RoboDK station: main for aircraftCOPY.rdk

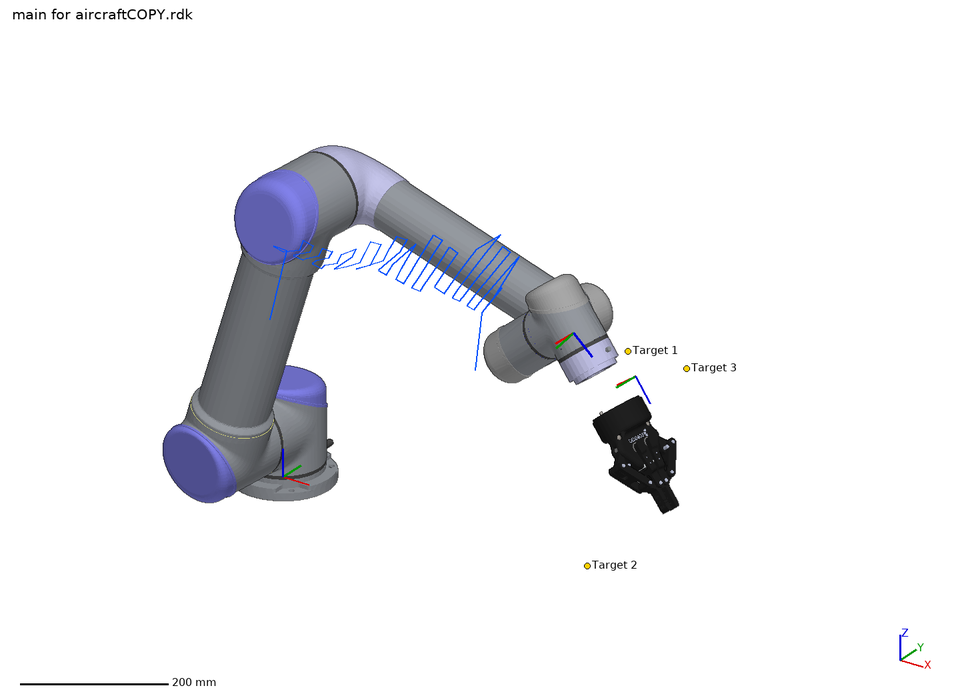
[picture v0: the station drawn from its stored meshes, robots at their saved joint values, targets as dots, program paths as lines]
Station main. Poses are relative to the parent item; angles as X-Y-Z fixed-axis rotations.
  - frame UR5 Base at (0, 0, 0) mm
    - robot UR5: 6 axes, payload 5 kg, reach 850 mm, repeatability 0.1 mm, weight 18.4 kg
        modified DH rows (alpha deg, a mm, theta deg, d mm): 0, 0, 0, 89.2; 90, 0, 180, 0; 0, 425, 0, 0; 0, 392.43, 0, 109; -90, 0, 0, 93.65; 90, 0, 180, 82
        joint limits [-360, -360, -360, -360, -360, -360] to [360, 360, 360, 360, 360, 360]; home [0, -90, -90, 0, 90, 0]; saved at [-4.126, -107.813, -86.6, -35.896, 88.406, -3.183]
      - tool Gripper RobotiQ 85 Fully closed, TCP at (0, 0, 266.2) mm, size 121.5 x 75 x 160.2 mm
      - frame Object at (8, -67.5, 31) mm
    - target Target 1 (Cartesian target) at (643.45, -109, 411.64) mm, rotated rx -90 ry 0 rz -90 deg; joints [0, -86.624, -123.251, 29.876, 90, 0] of UR5
    - target Target 2 (Cartesian target) at (575.78, -109, 70.86) mm, rotated rx -135 ry 0 rz -90 deg; joints [0, -90, -135, 0, 90, 0] of UR5
    - target Target 3 (Cartesian target) at (739.63, -109, 412.97) mm, rotated rx -105 ry 0 rz -90 deg; joints [0, -90, -105, 0, 90, 0] of UR5
    - frame Object at (559.36, -117, 419.3) mm, rotated rx -132.29 ry 0 rz -90 deg
      - object cloud_8 at (0, 0, 0) mm
  - program Path1 (108 instructions, listed below)
  - machining project Path1 settings: rotZ(0) | rotX(0)*rotY(0) | rotZ(0) | onStart | onPathStart | onApproach | onPoint | onRetract | onFinish | SetRPM(%1) | SetTool(%1) | Extruder(%1) | default | default | OutOnMov(%1) | OutOffMov(%1) | onPathFinish | M_RunCode(%1)
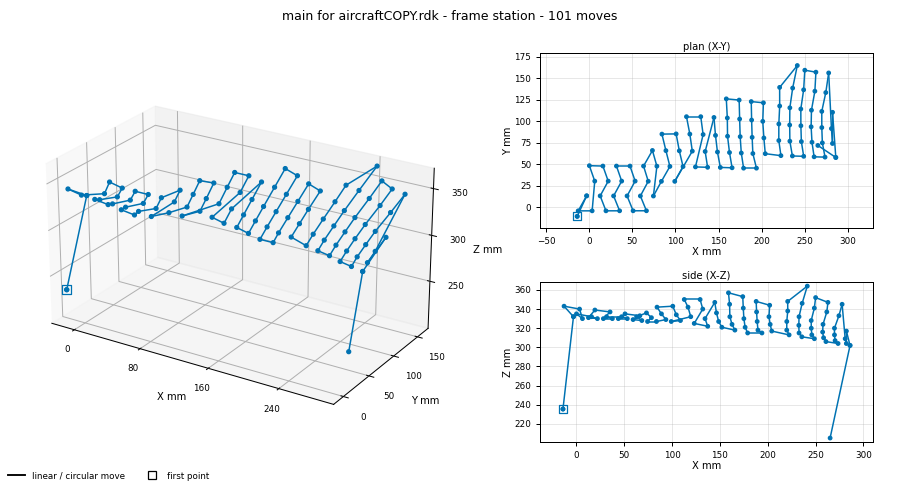
[picture p0: tool path of main for aircraftCOPY.rdk in frame station, 101 of 101 moves have a stored position in this frame; points joined in program order, loops and branches not executed]

--- program Path1 (robot UR5) ---
  Smooth(5)
  Set Ref.: UR5 Base
  Set Tool: Gripper RobotiQ 85 Fully closed
  Show Gripper RobotiQ 85 Fully closed
  Set speed (5.0 mm/s)
  MoveJ 1 to (-14.04, -10.4, 235.49) mm, rotated rx -13.93 ry 6.12 rz -1.51 deg; joints [4.658, -99.481, -81.097, -56.074, 81.119, 3.913]
  MoveL 2 to (-14.04, -10.4, 235.49) mm, rotated rx -13.93 ry 6.12 rz -1.51 deg; joints [4.658, -99.481, -81.097, -56.074, 81.119, 3.913]
  MoveL 3 to (-3.06, 13.38, 332) mm, rotated rx -13.93 ry 6.12 rz -1.51 deg; joints [3.175, -108.37, -82.037, -46.06, 81.936, 2.662]
  MoveL 4 to (-3.06, 13.38, 332) mm, rotated rx -13.93 ry 6.12 rz -1.51 deg; joints [3.175, -108.37, -82.037, -46.06, 81.936, 2.662]
  Set speed (5.0 mm/s)
  MoveL 5 to (-12.91, -4.04, 343) mm, rotated rx -32.27 ry 3.58 rz -2.26 deg; joints [2.431, -124.577, -46.301, -83.798, 85.122, 2.351]
  MoveL 6 to (3.3, -4, 340) mm, rotated rx -29.46 ry 5.28 rz -2.98 deg; joints [2.075, -121.423, -52.584, -77.822, 83.29, 1.983]
  MoveL 7 to (6.33, 30.48, 330) mm, rotated rx 2.3 ry 4.12 rz 0.17 deg; joints [1.192, -104.072, -102.448, -13.533, 84.96, 0.769]
  MoveL 8 to (0.08, 48.39, 335) mm, rotated rx 9.26 ry 5.03 rz 0.82 deg; joints [2.717, -105.068, -110.917, 2.753, 82.63, 1.494]
  MoveL 9 to (15.8, 47.96, 332) mm, rotated rx 8.64 ry 2.64 rz 0.4 deg; joints [-0.895, -105.14, -109.708, 1.212, 88.073, -0.496]
  MoveL 10 to (21.95, 30.48, 330) mm, rotated rx 1.48 ry 1.8 rz 0.05 deg; joints [-2.088, -104.786, -100.703, -15.298, 89.78, -1.364]
  MoveL 11 to (12.62, 13.34, 331) mm, rotated rx -12.78 ry 2.95 rz -0.67 deg; joints [-0.216, -108.437, -82.477, -44.133, 87.1, -0.177]
  MoveL 12 to (19.34, -3.99, 339) mm, rotated rx -27.21 ry 3.75 rz -1.93 deg; joints [-0.143, -119.939, -55.839, -73.653, 85.831, -0.134]
  MoveL 13 to (35.18, -3.97, 337) mm, rotated rx -25.88 ry 3.5 rz -1.7 deg; joints [-1.638, -119.083, -57.679, -71.257, 86.718, -1.522]
  MoveL 14 to (28.2, 13.3, 330) mm, rotated rx -11.29 ry 2.61 rz -0.52 deg; joints [-1.946, -108.209, -83.758, -41.541, 88.497, -1.566]
  MoveL 15 to (37.57, 30.48, 330) mm, rotated rx 1.89 ry 1.74 rz 0.06 deg; joints [-3.839, -105.297, -100.404, -14.689, 91.184, -2.488]
  MoveL 16 to (31.52, 47.96, 332) mm, rotated rx 6.96 ry 1.23 rz 0.15 deg; joints [-3.717, -105.465, -107.483, -2.398, 91.793, -2.15]
  MoveL 17 to (47.23, 47.96, 332) mm, rotated rx 8.92 ry 1.1 rz 0.17 deg; joints [-5.68, -106.487, -108.129, 1.171, 93.63, -3.127]
  MoveL 18 to (53.2, 30.48, 330) mm, rotated rx 3.33 ry 3.03 rz 0.18 deg; joints [-4.727, -105.67, -101.292, -11.942, 90.643, -2.971]
  MoveL 19 to (43.82, 13.3, 330) mm, rotated rx -9.75 ry 3.74 rz -0.64 deg; joints [-2.827, -107.971, -85.284, -38.649, 87.952, -2.229]
  MoveL 20 to (50.83, -3.94, 335) mm, rotated rx -26.54 ry 2.66 rz -1.33 deg; joints [-3.395, -120.113, -55.49, -73.063, 88.259, -3.166]
  MoveL 21 to (66.29, -3.92, 333) mm, rotated rx -26.5 ry 0.34 rz -0.17 deg; joints [-5.97, -121.072, -53.703, -74.084, 91.773, -5.567]
  MoveL 22 to (59.27, 13.26, 329) mm, rotated rx -8.2 ry 4.18 rz -0.6 deg; joints [-4.126, -107.813, -86.6, -35.896, 88.406, -3.183]
  MoveL 23 to (68.4, 30.3, 328) mm, rotated rx 4.71 ry 3.77 rz 0.31 deg; joints [-5.958, -105.952, -102.01, -9.54, 90.942, -3.631]
  MoveL 24 to (62.95, 47.96, 332) mm, rotated rx 11.37 ry 2.76 rz 0.56 deg; joints [-6.391, -107.482, -109.437, 5.996, 92.664, -3.283]
  MoveL 25 to (73.25, 66.03, 336) mm, rotated rx 17.27 ry 1.87 rz 0.58 deg; joints [-8.642, -111.204, -114.03, 20.082, 95.874, -3.664]
  MoveL 26 to (78.43, 47.81, 331) mm, rotated rx 12.53 ry 3.11 rz 0.69 deg; joints [-7.991, -108.278, -109.451, 7.928, 93.753, -3.968]
  MoveL 27 to (74.39, 13.18, 327) mm, rotated rx -4.76 ry 3.26 rz -0.27 deg; joints [-6.351, -107.433, -89.554, -29.969, 91.059, -4.644]
  MoveL 28 to (83.67, 30.21, 327) mm, rotated rx 6.61 ry 3.96 rz 0.46 deg; joints [-7.59, -106.614, -102.837, -6.179, 92.179, -4.424]
  MoveL 29 to (93.53, 47.52, 329) mm, rotated rx 13.66 ry 4.79 rz 1.16 deg; joints [-8.579, -108.731, -109.835, 9.966, 92.601, -4.11]
  MoveL 30 to (88.89, 65.84, 335) mm, rotated rx 18.59 ry 2.63 rz 0.88 deg; joints [-10.002, -112.249, -113.92, 22.315, 96.386, -4.032]
  MoveL 31 to (84.27, 85.02, 342) mm, rotated rx 19.46 ry 0.64 rz 0.23 deg; joints [-11.204, -114.4, -115.675, 26.899, 99.636, -4.386]
  MoveL 32 to (100.76, 85.27, 343) mm, rotated rx 22.25 ry 2.56 rz 1.05 deg; joints [-11.8, -116.671, -116.019, 32.433, 98.32, -4.065]
  MoveL 33 to (104.44, 65.64, 334) mm, rotated rx 20.16 ry 4.48 rz 1.64 deg; joints [-10.489, -113.289, -114.187, 25.277, 94.948, -3.958]
  MoveL 34 to (108.77, 47.38, 328) mm, rotated rx 15.72 ry 6.99 rz 1.96 deg; joints [-8.804, -109.718, -110.698, 13.955, 90.618, -3.942]
  MoveL 35 to (99.15, 30.21, 327) mm, rotated rx 8.68 ry 5.48 rz 0.83 deg; joints [-8.36, -107.362, -103.956, -2.166, 91.429, -4.622]
  MoveL 36 to (119.53, 65.25, 332) mm, rotated rx 21.76 ry 7.28 rz 2.9 deg; joints [-10.132, -114.088, -114.701, 28.264, 91.652, -3.57]
  MoveL 37 to (116.65, 85.02, 342) mm, rotated rx 23.97 ry 4.72 rz 2.09 deg; joints [-12.039, -117.925, -116.146, 35.627, 96.264, -3.799]
  MoveL 38 to (112.76, 105.23, 350) mm, rotated rx 22.75 ry 2.4 rz 1.01 deg; joints [-13.632, -119.241, -116.861, 36.235, 100.237, -4.599]
  MoveL 39 to (129.32, 105.23, 350) mm, rotated rx 25.49 ry 5.83 rz 2.77 deg; joints [-12.898, -121.304, -117.349, 41.728, 95.891, -3.75]
  MoveL 40 to (132.07, 84.52, 340) mm, rotated rx 25.16 ry 7.46 rz 3.49 deg; joints [-11.683, -118.575, -116.325, 37.699, 92.926, -3.469]
  MoveL 41 to (123.16, 46.95, 325) mm, rotated rx 17.31 ry 8.78 rz 2.72 deg; joints [-9.209, -110.364, -111.216, 16.734, 89.155, -3.906]
  MoveL 42 to (137.27, 46.51, 322) mm, rotated rx 18.11 ry 9.74 rz 3.17 deg; joints [-10.188, -110.797, -111.09, 17.851, 89.059, -4.198]
  MoveL 43 to (134.43, 64.85, 330) mm, rotated rx 21.94 ry 8.91 rz 3.57 deg; joints [-10.654, -114.25, -114.327, 28.246, 90.392, -3.735]
  MoveL 44 to (144.64, 104.33, 347) mm, rotated rx 27.45 ry 6.48 rz 3.35 deg; joints [-14.285, -122.842, -116.779, 44.62, 96.51, -3.692]
  MoveL 45 to (146.42, 83.53, 336) mm, rotated rx 26.11 ry 8.64 rz 4.21 deg; joints [-12.502, -119.014, -116.077, 38.811, 92.396, -3.528]
  MoveL 46 to (148.69, 64.26, 327) mm, rotated rx 21.87 ry 9.27 rz 3.7 deg; joints [-12.115, -114.309, -113.603, 27.514, 91.369, -4.26]
  MoveL 47 to (152.04, 46.37, 321) mm, rotated rx 18.81 ry 9.71 rz 3.29 deg; joints [-11.955, -111.655, -110.45, 18.745, 90.723, -4.788]
  MoveL 48 to (165.67, 45.93, 318) mm, rotated rx 18.23 ry 9.46 rz 3.1 deg; joints [-13.74, -111.641, -109.321, 17.009, 92.603, -5.619]
  MoveL 49 to (162.66, 63.67, 324) mm, rotated rx 22.01 ry 9.27 rz 3.72 deg; joints [-13.823, -114.576, -112.803, 27.09, 92.981, -4.826]
  MoveL 50 to (160.39, 82.53, 332) mm, rotated rx 26.15 ry 8.57 rz 4.18 deg; joints [-14.321, -119.011, -115.28, 38.024, 94.217, -4.029]
  MoveL 51 to (160.14, 103.73, 345) mm, rotated rx 29.01 ry 7.31 rz 4.04 deg; joints [-15.477, -124.202, -116.052, 46.772, 96.704, -3.605]
  MoveL 52 to (158.95, 125.93, 357) mm, rotated rx 25.77 ry 6.33 rz 3.05 deg; joints [-16.373, -124.524, -116.673, 44.444, 98.668, -4.696]
  MoveL 53 to (173.88, 124.52, 353) mm, rotated rx 25.79 ry 10.53 rz 5.05 deg; joints [-14.709, -123.729, -117.264, 44.369, 92.422, -4.254]
  MoveL 54 to (174.43, 102.53, 341) mm, rotated rx 29.39 ry 9.23 rz 5.16 deg; joints [-15.613, -124.047, -115.912, 46.829, 94.645, -3.565]
  MoveL 55 to (175.05, 82.04, 330) mm, rotated rx 26.13 ry 8.93 rz 4.35 deg; joints [-15.808, -119.248, -114.366, 37.298, 95.246, -4.456]
  MoveL 56 to (176.35, 63.08, 321) mm, rotated rx 21.27 ry 8.37 rz 3.24 deg; joints [-16.144, -114.531, -111.386, 24.811, 96.094, -5.818]
  MoveL 57 to (179.02, 45.5, 315) mm, rotated rx 17.33 ry 7.76 rz 2.41 deg; joints [-16.496, -111.814, -107.484, 14.249, 96.84, -6.975]
  MoveL 58 to (193.93, 45.5, 315) mm, rotated rx 15.83 ry 5.39 rz 1.53 deg; joints [-19.64, -112.544, -104.549, 10.067, 101.967, -8.828]
  MoveL 59 to (189.76, 62.49, 318) mm, rotated rx 20.07 ry 7.01 rz 2.55 deg; joints [-18.678, -114.416, -109.502, 21.397, 99.823, -7.106]
  MoveL 60 to (188.94, 81.29, 327) mm, rotated rx 24.51 ry 8.87 rz 4.02 deg; joints [-17.525, -118.312, -113.096, 33.447, 96.94, -5.406]
  MoveL 61 to (188.34, 101.33, 337) mm, rotated rx 28.37 ry 10.38 rz 5.56 deg; joints [-16.395, -122.948, -115.43, 44.227, 94.131, -4.042]
  MoveL 62 to (187.89, 122.75, 348) mm, rotated rx 25.98 ry 12.27 rz 5.91 deg; joints [-15.025, -123.348, -117.013, 43.906, 90.8, -4.333]
  MoveL 63 to (202.02, 121.34, 344) mm, rotated rx 26.28 ry 11.02 rz 5.39 deg; joints [-17.837, -123.694, -115.725, 43.214, 94.876, -5.018]
  MoveL 64 to (201.26, 99.82, 332) mm, rotated rx 27.33 ry 10.65 rz 5.46 deg; joints [-17.822, -121.884, -114.696, 41.39, 95.245, -4.702]
  MoveL 65 to (202.54, 80.55, 324) mm, rotated rx 22.52 ry 9.94 rz 4.09 deg; joints [-18.273, -117.028, -112.036, 29.179, 96.45, -6.232]
  MoveL 66 to (204.17, 62.3, 317) mm, rotated rx 18.16 ry 8.15 rz 2.66 deg; joints [-19.337, -113.803, -108.009, 17.452, 99.078, -7.939]
  MoveL 67 to (222.34, 60.03, 313) mm, rotated rx 14.21 ry 10.15 rz 2.56 deg; joints [-19.65, -112.166, -105.317, 9.466, 96.895, -9.244]
  MoveL 68 to (219.87, 77.55, 318) mm, rotated rx 18.99 ry 11.07 rz 3.78 deg; joints [-19.319, -114.796, -109.944, 21.46, 96.054, -7.674]
  MoveL 69 to (219.9, 96.77, 327) mm, rotated rx 25.69 ry 11.78 rz 5.61 deg; joints [-19.141, -120.51, -113.4, 37.111, 95.29, -5.582]
  MoveL 70 to (220.9, 117.63, 338) mm, rotated rx 27.73 ry 10.98 rz 5.72 deg; joints [-20.124, -124.595, -114.319, 44.049, 97.089, -5.184]
  MoveL 71 to (220.84, 139.23, 348) mm, rotated rx 31.61 ry 8.27 rz 5.06 deg; joints [-22.652, -130.842, -113.821, 53.503, 102.558, -4.337]
  MoveL 72 to (241.33, 164.59, 364) mm, rotated rx 35.26 ry 21.55 rz 14.56 deg; joints [-13.058, -135.826, -115.512, 62.282, 77.077, -2.264]
  MoveL 73 to (235.95, 138.43, 346) mm, rotated rx 31.94 ry 10.5 rz 6.48 deg; joints [-22.483, -130.861, -113.54, 53.548, 99.763, -4.227]
  MoveL 74 to (232.69, 115.54, 332) mm, rotated rx 28.97 ry 12.2 rz 6.68 deg; joints [-20.555, -124.887, -114.124, 45.319, 96.085, -4.911]
  MoveL 75 to (232.5, 95.59, 323) mm, rotated rx 24.2 ry 12.01 rz 5.34 deg; joints [-20.468, -119.484, -112.318, 33.541, 96.302, -6.46]
  MoveL 76 to (232.71, 76.82, 315) mm, rotated rx 17.53 ry 11.11 rz 3.48 deg; joints [-20.671, -114.346, -108.378, 17.969, 97.14, -8.681]
  MoveL 77 to (235.64, 59.65, 311) mm, rotated rx 12.24 ry 10.4 rz 2.24 deg; joints [-20.74, -111.961, -103.23, 5.235, 97.351, -10.365]
  MoveL 78 to (248.75, 59.26, 309) mm, rotated rx 12.05 ry 9.71 rz 2.06 deg; joints [-22.542, -112.61, -101.691, 3.921, 99.584, -11.351]
  MoveL 79 to (246.05, 76.33, 313) mm, rotated rx 16.26 ry 10.32 rz 2.99 deg; joints [-22.593, -114.428, -106.368, 14.602, 99.578, -9.94]
  MoveL 80 to (245.49, 94.7, 320) mm, rotated rx 22.41 ry 11.51 rz 4.7 deg; joints [-22.316, -118.687, -110.672, 29.268, 98.548, -7.676]
  MoveL 81 to (245.42, 114.15, 328) mm, rotated rx 28.59 ry 12.25 rz 6.59 deg; joints [-22.065, -124.555, -113.171, 43.627, 97.517, -5.409]
  MoveL 82 to (248.69, 136.43, 341) mm, rotated rx 30.93 ry 11.5 rz 6.81 deg; joints [-23.225, -129.548, -113.211, 50.878, 99.389, -4.786]
  MoveL 83 to (250.04, 159.16, 352) mm, rotated rx 26.25 ry 18.79 rz 9.03 deg; joints [-17.787, -127.605, -116.462, 47.664, 86.247, -5.294]
  MoveL 84 to (262.92, 156.9, 347) mm, rotated rx 21.2 ry 15.74 rz 6.01 deg; joints [-21.942, -124.051, -114.454, 37.527, 93.638, -8.034]
  MoveL 85 to (261.72, 134.83, 337) mm, rotated rx 31 ry 11.54 rz 6.85 deg; joints [-24.728, -129.529, -112.168, 49.83, 100.814, -5.073]
  MoveL 86 to (257.76, 112.76, 324) mm, rotated rx 27.1 ry 12.19 rz 6.17 deg; joints [-23.593, -123.475, -112.082, 39.969, 99.09, -6.354]
  MoveL 87 to (257.38, 93.52, 316) mm, rotated rx 20.85 ry 12.11 rz 4.57 deg; joints [-23.182, -117.732, -109.535, 25.67, 98.637, -8.55]
  MoveL 88 to (258.36, 75.6, 310) mm, rotated rx 14.7 ry 11.57 rz 3.01 deg; joints [-22.947, -113.864, -105.096, 11.402, 98.422, -10.624]
  MoveL 89 to (260.82, 58.69, 306) mm, rotated rx 11.48 ry 10.6 rz 2.14 deg; joints [-23.175, -112.649, -100.685, 2.498, 99.145, -11.851]
  MoveL 90 to (273.51, 58.3, 304) mm, rotated rx 10.15 ry 11.57 rz 2.06 deg; joints [-23.693, -112.669, -99.127, -0.18, 98.385, -12.554]
  MoveL 91 to (270.4, 74.87, 307) mm, rotated rx 13.4 ry 11.33 rz 2.68 deg; joints [-24.269, -113.79, -103.28, 8.123, 99.653, -11.719]
  MoveL 92 to (269.75, 92.63, 313) mm, rotated rx 19.54 ry 12.42 rz 4.37 deg; joints [-24.263, -117.246, -108.159, 22.511, 99.222, -9.449]
  MoveL 93 to (269.73, 111.36, 320) mm, rotated rx 25.95 ry 12.08 rz 5.82 deg; joints [-25.067, -122.725, -110.92, 36.872, 100.629, -7.22]
  MoveL 94 to (274.38, 133.23, 333) mm, rotated rx 32.33 ry 11.69 rz 7.31 deg; joints [-26.013, -130.482, -111.059, 50.918, 101.818, -4.774]
  MoveL 95 to (277.73, 156, 345) mm, rotated rx 16.02 ry 10.84 rz 3.09 deg; joints [-26.843, -121.881, -110.129, 25.286, 102.813, -11.95]
  MoveL 96 to (280.94, 91.44, 309) mm, rotated rx 17.97 ry 12.11 rz 3.89 deg; joints [-25.625, -116.644, -106.509, 18.613, 100.652, -10.61]
  MoveL 97 to (282.15, 74.13, 304) mm, rotated rx 12.59 ry 11.89 rz 2.63 deg; joints [-25.048, -113.779, -102.009, 6.089, 99.639, -12.391]
  MoveL 98 to (282.21, 110.32, 317) mm, rotated rx 25.69 ry 12.39 rz 5.89 deg; joints [-26.213, -122.71, -109.865, 35.49, 101.381, -7.676]
  MoveL 99 to (286.01, 57.92, 302) mm, rotated rx 8.38 ry 11.9 rz 1.74 deg; joints [-24.523, -112.802, -96.959, -3.897, 98.433, -13.603]
  Set speed (5.0 mm/s)
  MoveL 100 to (286.01, 57.92, 302) mm, rotated rx 8.38 ry 11.9 rz 1.74 deg; joints [-24.523, -112.802, -96.959, -3.897, 98.433, -13.603]
  MoveL 101 to (265.18, 71.86, 205.19) mm, rotated rx 8.38 ry 11.9 rz 1.74 deg; joints [-26.286, -99.656, -105.532, -8.627, 99.899, -14.595]
